FUNCTION_BLOCK Skill_Position_anfahren_erweitert	IMPLEMENTS I_Skill_Roboter  
VAR_INPUT
	eSysCommand					:eSystemCommand; 						// Systembefehl an Skill
	eSysState					:eSystemState;							// Momentaner Zustand des Systems
	eObjState					:eObjectAktorState; 							// Momentaner Zustand des Objektes
	
	bLimit						:BOOL;
	bErreicht					:BOOL;
END_VAR
VAR_OUTPUT
	eSkillCommand				:eSkillCommand;							// Skillbefehl für Objekt
	eProzessvariable			:sRoboterProzessVariablen;				// Prozessvariablen für Objekt
	iErrorID					:INT;									// Fehlercode für System
END_VAR
VAR
	// Managementvariablen
	iState				:eSkillState;									// Information über Zustand von Skill
	
	// Managementvariablen 
	bGestartet			:BOOL;
	bGestoppt			:BOOL;
	
	// Zustandsvariablen
	bStarten			:BOOL;
	bStoppen			:BOOL;
	bObjektFertig		:BOOL;
	bWertErreicht		:BOOL;				
	bLimitErreicht		:BOOL;				
	bSkillFertig		:BOOL;
	bFehler				:BOOL;
	bResetten			:BOOL;
END_VAR

// Fehlerüberwachung
IF bFehler THEN
	iState := 3;
END_IF

//_______________________________________________________________
// Reaktion auf Input-Variablen:
	// Stoppen
	IF eSysCommand = 3 THEN
		bStoppen := M_Stop();
	ELSE 
		bStoppen := FALSE;
	END_IF

	// Resetten 
	IF eSysCommand = 4 THEN
		bResetten := M_Reset();
	ELSE
		bResetten := FALSE;
	END_IF
	
	// Limit
	IF bLimit THEN
		bLimitErreicht := M_Stop();
	ELSE
		bLimitErreicht := FALSE;
	END_IF
	
	// Erreicht
	IF bErreicht THEN
		bWertErreicht := M_Stop();
	ELSE
		bWertErreicht := FALSE;
	END_IF
//_______________________________________________________________
// Zustandsmanagement
CASE iState OF 
0: 	// BEREIT	
		// DO
		IF eObjState = 3 THEN		// Objekt wurde eingeschalten
			bStarten := TRUE;
		END_IF
		
		// TRANSITION
		IF bStarten	 THEN		
			bStarten := FALSE;
			eSkillCommand := 0;
			iState := 1;	
		END_IF
		
		
// _________________________________________________________________________________________________________________________
1: 	// LAUFEND
		// DO			
			// Stoppen durch Sysezm
			IF bStoppen THEN																								// Transition wenn System das Orbjekt stoppt
				bGestoppt := TRUE;
			END_IF
			
			// Objekt hat sich selber gestoppt
			IF eObjState = 4 THEN																							// Objekt hat Prozess abgeschlossen
				bObjektFertig := TRUE;																							// Objekt ist fertig und wieder bereit
			END_IF
			
		// TRANSITION 
		IF bGestoppt THEN																								// Transition zu BEREIT
			bGestoppt := FALSE;		
			eSkillCommand := 0;																					
			iState := 0;
		END_IF
		
		IF bObjektFertig THEN																							// Transition zu ABGESCHLOSSEN
			bObjektFertig := FALSE;																							// Skill wird nicht mehr ausgeführt
			iState := 2;																									// Objekt ist fertig und wieder bereit
		END_IF
		
		IF bLimitErreicht AND eObjState = 5 THEN																							// Transition zu LIMIT
			eSkillCommand := 0;	
			iState := 4;
		END_IF
		
		IF bWertErreicht AND eObjState = 5 THEN																							// Transition zu ERREICHT
			eSkillCommand := 0;	
			iState := 5;
		END_IF
			
// _________________________________________________________________________________________________________________________			
2: 	// ABGESCHLOSSEN
		// DO
		IF eObjState = 1 THEN																							// Objekt wurde geresettet
			bSkillFertig := TRUE;									
		END_IF
			
		//  TRANSITION
		IF bSkillFertig THEN
			bSkillFertig := FALSE;																																											// Resetten von Objekt
			iState := 0;
		END_IF
		
// _________________________________________________________________________________________________________________________
3: 	// FEHLER
		// DO 	
		
		// TRANSITION
		IF bResetten THEN
			iState := 0;
		END_IF
		
// _________________________________________________________________________________________________________________________			
4: 	// LIMIT
		// DO		
		M_Reset();
		
		IF eObjState = 1 THEN																								// Objekt wurde geresettet
			bResetten := TRUE;								
		END_IF
	
		// TRANSITION
		IF bResetten THEN
			bResetten := FALSE;
			eSkillCommand := 0;
			iState := 0;
		END_IF
			
// _________________________________________________________________________________________________________________________
5: 	// ERREICHT		
		// DO 
		M_Reset();
		
		IF eObjState = 1 THEN																							// Objekt wurde geresettet
			bSkillFertig := TRUE;									
		END_IF
		
		// TRANSITION
		IF bSkillFertig THEN
			bSkillFertig := FALSE;
			eSkillCommand := 0;
			iState := 0;
		END_IF
		
END_CASE

METHOD M_Reset : BOOL
eSkillCommand := 3;

IF eSkillCommand = 3 THEN
	M_Reset := TRUE;
ELSE
	M_Reset := FALSE;
END_IF
END_METHOD

METHOD M_Start : BOOL
// Prüfen von Bedingungen
	// Ist das  System im korrekten Status
	IF eSysState = 1 THEN
		// Ist der Skill im korrekten Status 
		IF iState = 0 THEN
			// Prüfen auf Fehler (Muss ergänzt werden)
				eSkillCommand := 1;	
		END_IF
	END_IF

IF eSkillCommand = 1 THEN
	M_Start := TRUE;
ELSE
	M_Start := FALSE;
END_IF
END_METHOD

METHOD M_Stop : BOOL
eSkillCommand := 2;

IF eSkillCommand = 2 THEN
	M_Stop := TRUE;
ELSE
	M_Stop := FALSE;
END_IF
END_METHOD

PROPERTY P_Prozessparameter : sRoboterProzessVariablen
SET
eProzessvariable := P_Prozessparameter;
END_SET
END_PROPERTY

PROPERTY P_State : eSkillState
GET
P_State := iState;
END_GET
END_PROPERTY

END_FUNCTION_BLOCK

(* stored: Version 1.1.0.1
   POU Skill_Position_anfahren_erweitert: Id {0faeff5c-0f03-4aac-baad-74d21fa33f42}, SpecialFunc None
   Method M_Reset: Id {90a4a0e6-4f25-4388-a676-3de2cdd8719a}
   Method M_Start: Id {c462b91c-21ad-4c34-889f-5080f62aa886}
   Method M_Stop: Id {cb09df2e-2836-4d32-9461-ebad67f043b9}
   Property P_Prozessparameter: Id {63af0c77-9f9e-4476-9d02-71fe5537f00e}
   Set Set: Id {7cf45128-fb11-4611-8d3b-f112736e31ef}
   Property P_State: Id {b3867011-d9c4-4d62-b060-41996585080e}
   Get Get: Id {b305b60a-91af-4c24-abe8-2cbacd874c26} *)
